# EPICS autosave request: support/optics/2-6-1/opticsApp/Db/xia_slit.req
$(P)$(HSC)hID
$(P)$(HSC)vID
$(P)$(HSC)hOrient
$(P)$(HSC)vOrient
$(P)$(HSC)enable
